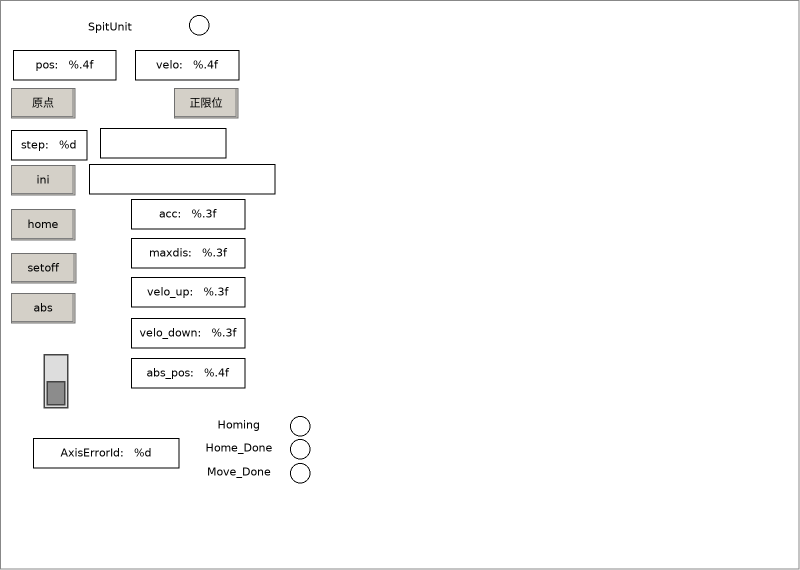
VISUALIZATION VIS_SpitUnit  // 800x570
    Button (11,209 64x31), "home", colour toggle: GVL_API.stSpitUnit.HomeExe
        toggle GVL_API.stSpitUnit.HomeExe
    Button (11,88 64x30), "原点", colour toggle: Axis[4].IO.snHome
        toggle Axis[4].IO.snHome
    Button (174,88 64x30), "正限位", colour toggle: Axis[4].IO.snLimitP
        toggle Axis[4].IO.snLimitP
    Rectangle (13,50 103x30), "pos: %.4f", text variable: Axis[4].Ref.NcToPlc.ActPos
    Rectangle (135,50 104x30), "velo: %.4f", text variable: Axis[4].Ref.NcToPlc.ActVelo
    Ellipse (189,15 20x20), colour toggle: Axis[4].Ref.Status.ControlLoopClosed
    Button (11,293 64x30), "abs", colour toggle: GVL_API.stSpitUnit.MoveAbsoluteExe
        toggle GVL_API.stSpitUnit.MoveAbsoluteExe
    Button (11,165 64x30), "ini", colour toggle: GVL_API.stSpitUnit.Initialize
        toggle GVL_API.stSpitUnit.Initialize
    Rectangle (131,358 114x30), "abs_pos: %.4f", text variable: GVL_API.stSpitUnit.target_position
        OnMouseDown: write GVL_API.stSpitUnit.target_position via Default
    Rectangle (131,277 114x30), "velo_up: %.3f", text variable: GVL_API.stSpitUnit.moving_speed_up
        OnMouseDown: write GVL_API.stSpitUnit.moving_speed_up via Default
    Rectangle (11,130 76x30), "step: %d", text variable: P_SpitUnit.SysStep
        OnMouseDown: write P_SpitUnit.SysStep via Default
    Button (11,253 65x30), "setoff", colour toggle: GVL_API.stSpitUnit.SetOff
        toggle GVL_API.stSpitUnit.SetOff
    Rectangle (100,128 126x30), text list: 'TextListSpitUnitState', text index: GVL_API.stSpitUnit.state
    Rectangle (89,164 186x30), text list: 'TextListSpitUnitErrorid', text index: GVL_API.stSpitUnit.error_code
    Label (70,12 80x30), "SpitUnit"
    Rectangle (33,438 146x30), "AxisErrorId: %d", text variable: GVL_API.stSpitUnit.AxisErrorId
    Rectangle (131,238 114x30), "maxdis: %.3f", text variable: GVL_API.stSpitUnit.spindle_length
        OnMouseDown: write GVL_API.stSpitUnit.spindle_length via Default
    Rectangle (131,199 114x30), "acc: %.3f", text variable: GVL_API.stSpitUnit.acceleration
        OnMouseDown: write GVL_API.stSpitUnit.acceleration via Default
    Rectangle (131,318 114x30), "velo_down: %.3f", text variable: GVL_API.stSpitUnit.moving_speed_down
        OnMouseDown: write GVL_API.stSpitUnit.moving_speed_down via Default
    Label (199,433 80x30), "Home_Done"
    Ellipse (290,439 20x20), colour toggle: GVL_API.stSpitUnit.Home_Done
    Label (199,457 80x30), "Move_Done"
    Ellipse (290,463 20x20), colour toggle: GVL_API.stSpitUnit.Move_Done
    DipSwitch (29,354 54x54), variable: GVL.HMI_btEmstop, behaviour: TOGGLE, style: Switch-DipSwitch-Gray
    Label (199,410 80x30), "Homing"
    Ellipse (290,416 20x20), colour toggle: GVL_API.stSpitUnit.Homing
END_VISUALIZATION

(* stored: Version 1.1.0.1, ProductVersion 3.1.4024.11
   Visu VIS_SpitUnit: Id {4e5bb5d8-3974-4dd4-b6d1-6f14444508fb} *)
